FUNCTION_BLOCK F_TIME_WEIGHTED_MEAN_LREAL (* Stores arriving data and releases the time weighted mean since the last GET event upon every GET event. *)
  (* Standard: 61499-2; Description: Stores arriving data and releases the time weighted mean since the last GET event upon every GET event. The elapsed time between values is determined via the time stamp. *)
  (* Version 1.0, 2017-06-13, Marc Jakobi, HTW Berlin *)
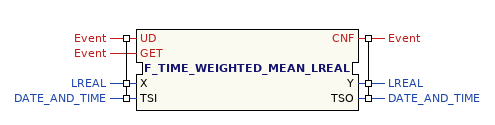
  EVENT_INPUT
    UD WITH X, TSI; (* Normal Execution Request *)
    GET;
  END_EVENT
  EVENT_OUTPUT
    CNF WITH Y, TSO; (* New average arrived *)
  END_EVENT
  VAR_INPUT
    X : LREAL; (* Input data *)
    TSI : DATE_AND_TIME; (* Time stamp *)
  END_VAR
  VAR_OUTPUT
    Y : LREAL; (* N minute mean of X *)
    TSO : DATE_AND_TIME; (* Time stamp *)
  END_VAR
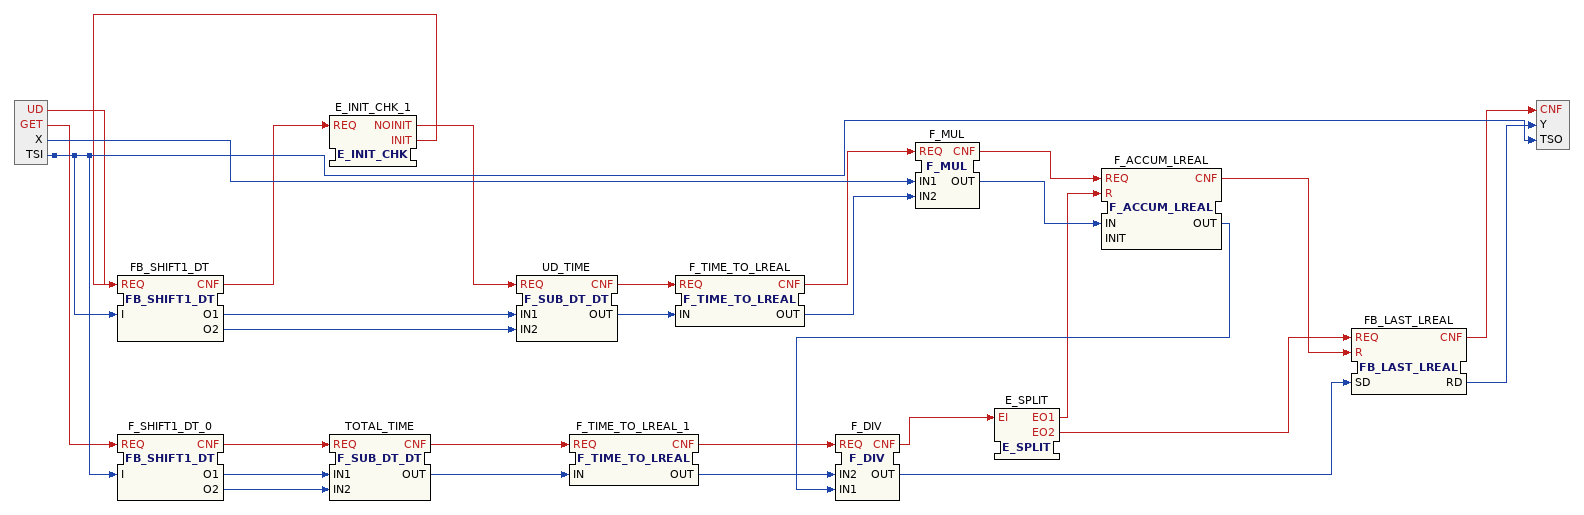
  FBS
    FB_SHIFT1_DT : FB_SHIFT1_DT;
    UD_TIME : F_SUB_DT_DT;
    F_TIME_TO_LREAL : F_TIME_TO_LREAL;
    F_SHIFT1_DT_0 : FB_SHIFT1_DT;
    TOTAL_TIME : F_SUB_DT_DT;
    F_TIME_TO_LREAL_1 : F_TIME_TO_LREAL;
    F_MUL : F_MUL;
    F_DIV : F_DIV;
    E_INIT_CHK_1 : E_INIT_CHK;
    F_ACCUM_LREAL : F_ACCUM_LREAL;
    E_SPLIT : E_SPLIT;
    FB_LAST_LREAL : FB_LAST_LREAL;
  END_FBS
  EVENT_CONNECTIONS
    UD_TIME.CNF TO F_TIME_TO_LREAL.REQ;
    GET TO F_SHIFT1_DT_0.REQ;
    F_SHIFT1_DT_0.CNF TO TOTAL_TIME.REQ;
    TOTAL_TIME.CNF TO F_TIME_TO_LREAL_1.REQ;
    F_TIME_TO_LREAL.CNF TO F_MUL.REQ;
    FB_SHIFT1_DT.CNF TO E_INIT_CHK_1.REQ;
    E_INIT_CHK_1.NOINIT TO UD_TIME.REQ;
    E_INIT_CHK_1.INIT TO FB_SHIFT1_DT.REQ;
    F_MUL.CNF TO F_ACCUM_LREAL.REQ;
    F_TIME_TO_LREAL_1.CNF TO F_DIV.REQ;
    F_DIV.CNF TO E_SPLIT.EI;
    E_SPLIT.EO1 TO F_ACCUM_LREAL.R;
    UD TO FB_SHIFT1_DT.REQ;
    E_SPLIT.EO2 TO FB_LAST_LREAL.REQ;
    F_ACCUM_LREAL.CNF TO FB_LAST_LREAL.R;
    FB_LAST_LREAL.CNF TO CNF;
  END_CONNECTIONS
  DATA_CONNECTIONS
    TSI TO FB_SHIFT1_DT.I;
    FB_SHIFT1_DT.O1 TO UD_TIME.IN1;
    FB_SHIFT1_DT.O2 TO UD_TIME.IN2;
    UD_TIME.OUT TO F_TIME_TO_LREAL.IN;
    TSI TO F_SHIFT1_DT_0.I;
    F_SHIFT1_DT_0.O1 TO TOTAL_TIME.IN1;
    F_SHIFT1_DT_0.O2 TO TOTAL_TIME.IN2;
    TOTAL_TIME.OUT TO F_TIME_TO_LREAL_1.IN;
    X TO F_MUL.IN1;
    F_TIME_TO_LREAL.OUT TO F_MUL.IN2;
    F_MUL.OUT TO F_ACCUM_LREAL.IN;
    F_TIME_TO_LREAL_1.OUT TO F_DIV.IN2;
    F_ACCUM_LREAL.OUT TO F_DIV.IN1;
    TSI TO TSO;
    F_DIV.OUT TO FB_LAST_LREAL.SD;
    FB_LAST_LREAL.RD TO Y;
  END_CONNECTIONS
END_FUNCTION_BLOCK
